SYSTEM TEST_SYS2 (* System Configuration for testing TEST_RES2 *)
  (* Standard: 61499-1 *)
  (* Version 0.1, 2005-05-17, JHC, Holobloc Inc, Changed UDP sockets 1025-6 to 1031-2 to work with WXP. *)
  (* Version 0.0, 2004-06-08, JHC, Rockwell Automation *)
  APPLICATION APP1
  END_APPLICATION
  DEVICE DEV1 : FRAME_DEVICE(GRID := [2,1], BOUNDS := [100,100,150,150])
    RESOURCE INPUTS : PANEL_RESOURCE
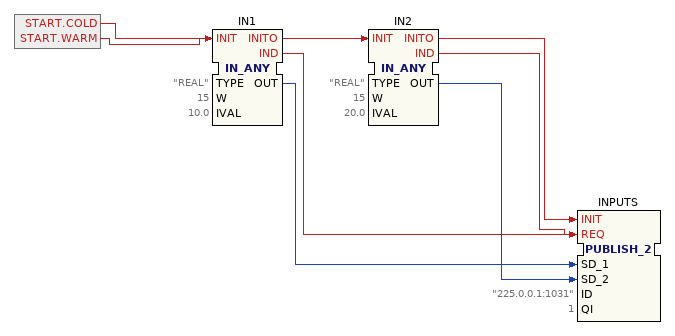
      FBS
        IN1 : IN_ANY(TYPE := "REAL", W := 15, IVAL := 10.0);
        IN2 : IN_ANY(TYPE := "REAL", W := 15, IVAL := 20.0);
        INPUTS : PUBLISH_2(ID := "225.0.0.1:1031", QI := 1);
      END_FBS
      EVENT_CONNECTIONS
        START.COLD TO IN1.INIT;
        START.WARM TO IN1.INIT;
        IN1.INITO TO IN2.INIT;
        IN2.INITO TO INPUTS.INIT;
        IN1.IND TO INPUTS.REQ;
        IN2.IND TO INPUTS.REQ;
      END_CONNECTIONS
      DATA_CONNECTIONS
        IN1.OUT TO INPUTS.SD_1;
        IN2.OUT TO INPUTS.SD_2;
      END_CONNECTIONS
    END_RESOURCE
    RESOURCE TESTED : TEST_RES2(INPUT_ID := "225.0.0.1:1031", OUTPUT_ID := "225.0.0.1:1032")
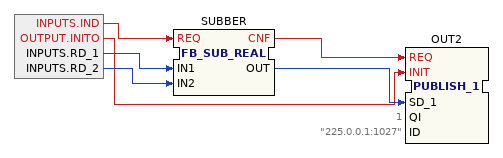
      FBS
        SUBBER : FB_SUB_REAL;
        OUT2 : PUBLISH_1(QI := 1, ID := "225.0.0.1:1027");
      END_FBS
      EVENT_CONNECTIONS
        INPUTS.IND TO SUBBER.REQ;
        SUBBER.CNF TO OUT2.REQ;
        OUTPUT.INITO TO OUT2.INIT;
      END_CONNECTIONS
      DATA_CONNECTIONS
        INPUTS.RD_1 TO SUBBER.IN1;
        INPUTS.RD_2 TO SUBBER.IN2;
        SUBBER.OUT TO OUT2.SD_1;
      END_CONNECTIONS
    END_RESOURCE
    RESOURCE OUTPUTS : PANEL_RESOURCE
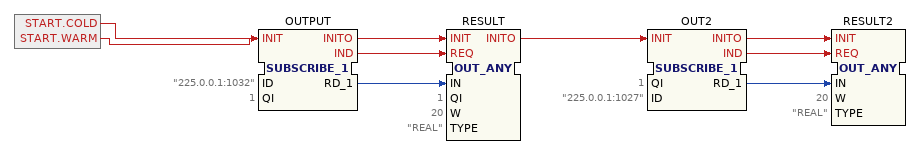
      FBS
        OUTPUT : SUBSCRIBE_1(ID := "225.0.0.1:1032", QI := 1);
        RESULT : OUT_ANY(QI := 1, W := 20, TYPE := "REAL");
        OUT2 : SUBSCRIBE_1(QI := 1, ID := "225.0.0.1:1027");
        RESULT2 : OUT_ANY(W := 20, TYPE := "REAL");
      END_FBS
      EVENT_CONNECTIONS
        START.COLD TO OUTPUT.INIT;
        START.WARM TO OUTPUT.INIT;
        OUTPUT.INITO TO RESULT.INIT;
        OUTPUT.IND TO RESULT.REQ;
        RESULT.INITO TO OUT2.INIT;
        OUT2.INITO TO RESULT2.INIT;
        OUT2.IND TO RESULT2.REQ;
      END_CONNECTIONS
      DATA_CONNECTIONS
        OUTPUT.RD_1 TO RESULT.IN;
        OUT2.RD_1 TO RESULT2.IN;
      END_CONNECTIONS
    END_RESOURCE
  END_DEVICE
END_SYSTEM
